{attribute 'pack_mode' := '1'} 
// ------------------------------------------------------------------------- 
//  SRCI Robot Library                                                
// ------------------------------------------------------------------------- 
//                                                                           
//  Object:      FreeDriveParCmd                                       
//  Author:      Thorsten Brach                                                
//  Date:        2024-06-22
//
//  Description:                                              
//   
//                                                                           
//  Copyright: 
//    (C) 2024 Thorsten Brach. All rights reserved                                                                                                                                            
//             Licensed under the MIT License.
//                                                                           
//  Disclaimer:                                                                           
//    This project is provided without any guarantee and can be used for   
//    private and commercial purposes. Any use is at the user’s 
//    own risk and responsibility.
//
// -------------------------------------------------------------------------
TYPE FreeDriveParCmd :
STRUCT
END_STRUCT
END_TYPE

{attribute 'pack_mode' := '1'} 
// ------------------------------------------------------------------------- 
//  SRCI Robot Library                                                
// ------------------------------------------------------------------------- 
//                                                                           
//  Object:      FreeDriveRecvData                                       
//  Author:      Thorsten Brach                                                
//  Date:        2024-06-22
//
//  Description:                                              
//   
//                                                                           
//  Copyright: 
//    (C) 2024 Thorsten Brach. All rights reserved                                                                                                                                            
//             Licensed under the MIT License.
//                                                                           
//  Disclaimer:                                                                           
//    This project is provided without any guarantee and can be used for   
//    private and commercial purposes. Any use is at the user’s 
//    own risk and responsibility.
//
// -------------------------------------------------------------------------
TYPE FreeDriveRecvData EXTENDS RspHeader :
STRUCT
  /// TRUE when function is exchanging data
  Enabled : BOOL;
END_STRUCT
END_TYPE

{attribute 'pack_mode' := '1'}
// ------------------------------------------------------------------------- 
//  SRCI Robot Library                                                
// ------------------------------------------------------------------------- 
//                                                                           
//  Object:      FreeDriveSendData                                       
//  Author:      Thorsten Brach                                                
//  Date:        2024-06-22
//
//  Description:                                              
//   
//                                                                           
//  Copyright: 
//    (C) 2024 Thorsten Brach. All rights reserved                                                                                                                                            
//             Licensed under the MIT License.
//                                                                           
//  Disclaimer:                                                                           
//    This project is provided without any guarantee and can be used for   
//    private and commercial purposes. Any use is at the user’s 
//    own risk and responsibility.
//
// -------------------------------------------------------------------------
TYPE FreeDriveSendData EXTENDS CmdHeader: 
STRUCT
  /// Set TRUE to activate "FreeDrive".
  Enable : BOOL;
END_STRUCT
END_TYPE

{attribute 'pack_mode' := '1'} 
// ------------------------------------------------------------------------- 
//  SRCI Robot Library                                                
// ------------------------------------------------------------------------- 
//                                                                           
//  Object:      MeasuringInputOutCmd                                       
//  Author:      Thorsten Brach                                                
//  Date:        2024-06-21
//
//  Description:                                              
//   
//                                                                           
//  Copyright: 
//    (C) 2024 Thorsten Brach. All rights reserved                                                                                                                                            
//             Licensed under the MIT License.
//                                                                           
//  Disclaimer:                                                                           
//    This project is provided without any guarantee and can be used for   
//    private and commercial purposes. Any use is at the user’s 
//    own risk and responsibility.
//
// -------------------------------------------------------------------------
TYPE MeasuringInputOutCmd :
STRUCT
  /// FB is returning a unique ID for the called measurement.
  MeasuringID        : UINT;
  /// Measured robot position value at the rising edge of the digital input in selected coordinate systems (see input parameters ToolNo and FrameNo).
  Measurings         : ARRAY[1..2] OF MeasuringInputResult;  
END_STRUCT
END_TYPE

{attribute 'pack_mode' := '1'} 
// ------------------------------------------------------------------------- 
//  SRCI Robot Library                                                
// ------------------------------------------------------------------------- 
//                                                                           
//  Object:      MeasuringInputParCmd                                       
//  Author:      Thorsten Brach                                                
//  Date:        2024-06-21
//
//  Description:                                              
//   
//                                                                           
//  Copyright: 
//    (C) 2024 Thorsten Brach. All rights reserved                                                                                                                                            
//             Licensed under the MIT License.
//                                                                           
//  Disclaimer:                                                                           
//    This project is provided without any guarantee and can be used for   
//    private and commercial purposes. Any use is at the user’s 
//    own risk and responsibility.
//
// -------------------------------------------------------------------------
TYPE MeasuringInputParCmd :
STRUCT
  /// Type of measurement (at least one option must be supported):
  MeasuringMode      : MeasuringIoMode;
  /// Specifies the desired digital input register. 
  /// More information about the different periphery register can be found in chapter 6.4
  Index              : USINT;
  ///Specifies the desired bit in the digital input register, that should be read. 
  /// More information about the different periphery register can be found in chapter 6.4.
  BitNumber          : USINT;
END_STRUCT
END_TYPE

{attribute 'pack_mode' := '1'} 
// ------------------------------------------------------------------------- 
//  SRCI Robot Library                                                
// ------------------------------------------------------------------------- 
//                                                                           
//  Object:      MeasuringInputRecvData                                       
//  Author:      Thorsten Brach                                                
//  Date:        2024-06-21
//
//  Description:                                              
//   
//                                                                           
//  Copyright: 
//    (C) 2024 Thorsten Brach. All rights reserved                                                                                                                                            
//             Licensed under the MIT License.
//                                                                           
//  Disclaimer:                                                                           
//    This project is provided without any guarantee and can be used for   
//    private and commercial purposes. Any use is at the user’s 
//    own risk and responsibility.
//
// -------------------------------------------------------------------------
TYPE MeasuringInputRecvData EXTENDS RspHeader :
STRUCT
  /// FB is returning a unique ID for the called measurement.
  MeasuringID        : UINT;
  /// Measured robot position value at the rising edge of the digital input in selected coordinate systems (see input parameters ToolNo and FrameNo).
  Measurings         : ARRAY[1..2] OF MeasuringInputResult;  
END_STRUCT
END_TYPE

{attribute 'pack_mode' := '1'}
// ------------------------------------------------------------------------- 
//  SRCI Robot Library                                                
// ------------------------------------------------------------------------- 
//                                                                           
//  Object:      MeasuringInputSendData                                       
//  Author:      Thorsten Brach                                                
//  Date:        2024-06-21
//
//  Description:                                              
//   
//                                                                           
//  Copyright: 
//    (C) 2024 Thorsten Brach. All rights reserved                                                                                                                                            
//             Licensed under the MIT License.
//                                                                           
//  Disclaimer:                                                                           
//    This project is provided without any guarantee and can be used for   
//    private and commercial purposes. Any use is at the user’s 
//    own risk and responsibility.
//
// -------------------------------------------------------------------------
TYPE MeasuringInputSendData EXTENDS CmdHeader:   
STRUCT
  /// Type of measurement (at least one option must be supported):
  MeasuringMode      : MeasuringIoMode;
  /// Specifies the desired digital input register. 
  /// More information about the different periphery register can be found in chapter 6.4
  Index              : USINT;
  ///Specifies the desired bit in the digital input register, that should be read. 
  /// More information about the different periphery register can be found in chapter 6.4.
  BitNumber          : USINT;
END_STRUCT
END_TYPE

{attribute 'pack_mode' := '1'} 
// ------------------------------------------------------------------------- 
//  SRCI Robot Library                                                
// ------------------------------------------------------------------------- 
//                                                                           
//  Object:      BrakeTestOutCmd                                       
//  Author:      Thorsten Brach                                                
//  Date:        2024-06-01
//
//  Description:                                              
//   
//                                                                           
//  Copyright: 
//    (C) 2024 Thorsten Brach. All rights reserved                                                                                                                                            
//             Licensed under the MIT License.
//                                                                           
//  Disclaimer:                                                                           
//    This project is provided without any guarantee and can be used for   
//    private and commercial purposes. Any use is at the user’s 
//    own risk and responsibility.
//
// -------------------------------------------------------------------------
TYPE OpenBrakeOutCmd :
STRUCT
  /// TRUE when "OpenBrake" is active.
  Enabled                   : BOOL;  
  /// Indicates the brake release status of the main robot axes.
  /// • TRUE: The brake of the axis is opened.
  /// • FALSE: The brake of the axis is closed.
  /// See Table 6-735 for bit assignment
  RobotAxesBrakeReleased    : RobotAxesFlags;
  /// Indicates the brake release status of the external robot axes.
  /// • TRUE: The brake of the axis is opened.
  /// • FALSE: The brake of the axis is closed/not supported
  /// See Table 6-735 for bit assignment
  ExternalAxesBrakeReleased : ExternalAxesFlags;
END_STRUCT
END_TYPE

{attribute 'pack_mode' := '1'} 
// ------------------------------------------------------------------------- 
//  SRCI Robot Library                                                
// ------------------------------------------------------------------------- 
//                                                                           
//  Object:      OpenBrakeParCmd                                       
//  Author:      Thorsten Brach                                                
//  Date:        2024-06-01
//
//  Description:                                              
//   
//                                                                           
//  Copyright: 
//    (C) 2024 Thorsten Brach. All rights reserved                                                                                                                                            
//             Licensed under the MIT License.
//                                                                           
//  Disclaimer:                                                                           
//    This project is provided without any guarantee and can be used for   
//    private and commercial purposes. Any use is at the user’s 
//    own risk and responsibility.
//
// -------------------------------------------------------------------------
TYPE OpenBrakeParCmd :
STRUCT
  /// Defines which brake of the robot axes must be released.
  /// • TRUE: Open the brake of the axis.
  /// • FALSE (default): Close the brake of the axis.
  RobotAxesBrakeRelease    : RobotAxesFlags;
  /// Defines which brake of the external robot axis must be released.
  /// • TRUE: Open the brake of the axis.
  /// • FALSE (default): Close the brake of the axis.
  /// See Table 6-676 for bit assignment.
  ExternalAxesBrakeRelease : ExternalAxesFlags;
END_STRUCT
END_TYPE

{attribute 'pack_mode' := '1'} 
// ------------------------------------------------------------------------- 
//  SRCI Robot Library                                                
// ------------------------------------------------------------------------- 
//                                                                           
//  Object:      BrakeTestRecvData                                       
//  Author:      Thorsten Brach                                                
//  Date:        2024-06-01
//
//  Description:                                              
//   
//                                                                           
//  Copyright: 
//    (C) 2024 Thorsten Brach. All rights reserved                                                                                                                                            
//             Licensed under the MIT License.
//                                                                           
//  Disclaimer:                                                                           
//    This project is provided without any guarantee and can be used for   
//    private and commercial purposes. Any use is at the user’s 
//    own risk and responsibility.
//
// -------------------------------------------------------------------------
TYPE OpenBrakeRecvData EXTENDS RspHeader :
STRUCT
  /// TRUE when "OpenBrake" is active.
  Enabled                   : BYTE;  
  /// Indicates the brake release status of the main robot axes.
  /// • TRUE: The brake of the axis is opened.
  /// • FALSE: The brake of the axis is closed.
  /// See Table 6-735 for bit assignment
  RobotAxesBrakeReleased    : BYTE;
  /// Indicates the brake release status of the external robot axes.
  /// • TRUE: The brake of the axis is opened.
  /// • FALSE: The brake of the axis is closed/not supported
  /// See Table 6-735 for bit assignment
  ExternalAxesBrakeReleased : BYTE;
END_STRUCT
END_TYPE

{attribute 'pack_mode' := '1'}
// ------------------------------------------------------------------------- 
//  SRCI Robot Library                                                
// ------------------------------------------------------------------------- 
//                                                                           
//  Object:      BrakeTestSendData                                       
//  Author:      Thorsten Brach                                                
//  Date:        2024-06-01
//
//  Description:                                              
//   
//                                                                           
//  Copyright: 
//    (C) 2024 Thorsten Brach. All rights reserved                                                                                                                                            
//             Licensed under the MIT License.
//                                                                           
//  Disclaimer:                                                                           
//    This project is provided without any guarantee and can be used for   
//    private and commercial purposes. Any use is at the user’s 
//    own risk and responsibility.
//
// -------------------------------------------------------------------------
TYPE OpenBrakeSendData EXTENDS CmdHeader:   
STRUCT
  /// Defines which brake of the robot axes must be released.
  /// • TRUE: Open the brake of the axis.
  /// • FALSE (default): Close the brake of the axis.
  RobotAxesBrakeRelease    : BYTE;
  /// Defines which brake of the external robot axis must be released.
  /// • TRUE: Open the brake of the axis.
  /// • FALSE (default): Close the brake of the axis.
  /// See Table 6-676 for bit assignment.
  ExternalAxesBrakeRelease : BYTE;
END_STRUCT
END_TYPE

{attribute 'pack_mode' := '1'} 
// ------------------------------------------------------------------------- 
//  SRCI Robot Library                                                
// ------------------------------------------------------------------------- 
//                                                                           
//  Object:      PathAccuracyModeOutCmd                                       
//  Author:      Thorsten Brach                                                
//  Date:        2024-06-22
//
//  Description:                                              
//   
//                                                                           
//  Copyright: 
//    (C) 2024 Thorsten Brach. All rights reserved                                                                                                                                            
//             Licensed under the MIT License.
//                                                                           
//  Disclaimer:                                                                           
//    This project is provided without any guarantee and can be used for   
//    private and commercial purposes. Any use is at the user’s 
//    own risk and responsibility.
//
// -------------------------------------------------------------------------
TYPE PathAccuracyModeOutCmd :
STRUCT
END_STRUCT
END_TYPE

{attribute 'pack_mode' := '1'} 
// ------------------------------------------------------------------------- 
//  SRCI Robot Library                                                
// ------------------------------------------------------------------------- 
//                                                                           
//  Object:      PathAccuracyModeParCmd                                       
//  Author:      Thorsten Brach                                                
//  Date:        2024-06-22
//
//  Description:                                              
//   
//                                                                           
//  Copyright: 
//    (C) 2024 Thorsten Brach. All rights reserved                                                                                                                                            
//             Licensed under the MIT License.
//                                                                           
//  Disclaimer:                                                                           
//    This project is provided without any guarantee and can be used for   
//    private and commercial purposes. Any use is at the user’s 
//    own risk and responsibility.
//
// -------------------------------------------------------------------------
TYPE PathAccuracyModeParCmd :
STRUCT
END_STRUCT
END_TYPE

{attribute 'pack_mode' := '1'} 
// ------------------------------------------------------------------------- 
//  SRCI Robot Library                                                
// ------------------------------------------------------------------------- 
//                                                                           
//  Object:      PathAccuracyModeRecvData                                       
//  Author:      Thorsten Brach                                                
//  Date:        2024-06-22
//
//  Description:                                              
//   
//                                                                           
//  Copyright: 
//    (C) 2024 Thorsten Brach. All rights reserved                                                                                                                                            
//             Licensed under the MIT License.
//                                                                           
//  Disclaimer:                                                                           
//    This project is provided without any guarantee and can be used for   
//    private and commercial purposes. Any use is at the user’s 
//    own risk and responsibility.
//
// -------------------------------------------------------------------------
TYPE PathAccuracyModeRecvData EXTENDS RspHeader :
STRUCT
  /// TRUE while PathAccuracyMode is active
  Enabled : BOOL;
END_STRUCT
END_TYPE

{attribute 'pack_mode' := '1'}
// ------------------------------------------------------------------------- 
//  SRCI Robot Library                                                
// ------------------------------------------------------------------------- 
//                                                                           
//  Object:      PathAccuracyModeSendData                                       
//  Author:      Thorsten Brach                                                
//  Date:        2024-06-22
//
//  Description:                                              
//   
//                                                                           
//  Copyright: 
//    (C) 2024 Thorsten Brach. All rights reserved                                                                                                                                            
//             Licensed under the MIT License.
//                                                                           
//  Disclaimer:                                                                           
//    This project is provided without any guarantee and can be used for   
//    private and commercial purposes. Any use is at the user’s 
//    own risk and responsibility.
//
// -------------------------------------------------------------------------
TYPE PathAccuracyModeSendData EXTENDS CmdHeader: 
STRUCT
  /// Set TRUE to activate monitoring of work areas
  Enable             : BOOL;
END_STRUCT
END_TYPE

{attribute 'pack_mode' := '1'} 
// ------------------------------------------------------------------------- 
//  SRCI Robot Library                                                
// ------------------------------------------------------------------------- 
//                                                                           
//  Object:      UnitMeasurementOutCmd                                       
//  Author:      Thorsten Brach                                                
//  Date:        2024-08-11
//
//  Description:                                              
//   
//                                                                           
//  Copyright: 
//    (C) 2024 Thorsten Brach. All rights reserved                                                                                                                                            
//             Licensed under the MIT License.
//                                                                           
//  Disclaimer:                                                                           
//    This project is provided without any guarantee and can be used for   
//    private and commercial purposes. Any use is at the user’s 
//    own risk and responsibility.
//
// -------------------------------------------------------------------------
TYPE ReadCallSubprogramCyclicOutCmd :
STRUCT
  /// Cyclic input data of subprogram
  Data : ARRAY[0..25] OF BYTE;
END_STRUCT
END_TYPE

{attribute 'pack_mode' := '1'} 
// ------------------------------------------------------------------------- 
//  SRCI Robot Library                                                
// ------------------------------------------------------------------------- 
//                                                                           
//  Object:      UnitMeasurementParCmd                                       
//  Author:      Thorsten Brach                                                
//  Date:        2024-08-11
//
//  Description:                                              
//   
//                                                                           
//  Copyright: 
//    (C) 2024 Thorsten Brach. All rights reserved                                                                                                                                            
//             Licensed under the MIT License.
//                                                                           
//  Disclaimer:                                                                           
//    This project is provided without any guarantee and can be used for   
//    private and commercial purposes. Any use is at the user’s 
//    own risk and responsibility.
//
// -------------------------------------------------------------------------
TYPE ReadCallSubprogramCyclicParCmd :
STRUCT
END_STRUCT
END_TYPE

{attribute 'pack_mode' := '1'} 
// ------------------------------------------------------------------------- 
//  SRCI Robot Library                                                
// ------------------------------------------------------------------------- 
//                                                                           
//  Object:      ShiftPositionOutCmd                                       
//  Author:      Thorsten Brach                                                
//  Date:        2024-06-22
//
//  Description:                                              
//   
//                                                                           
//  Copyright: 
//    (C) 2024 Thorsten Brach. All rights reserved                                                                                                                                            
//             Licensed under the MIT License.
//                                                                           
//  Disclaimer:                                                                           
//    This project is provided without any guarantee and can be used for   
//    private and commercial purposes. Any use is at the user’s 
//    own risk and responsibility.
//
// -------------------------------------------------------------------------
TYPE ShiftPositionOutCmd :
STRUCT
  /// Tool index
  TransformedPosition       : RobotCartesianPosition;  
END_STRUCT
END_TYPE

{attribute 'pack_mode' := '1'} 
// ------------------------------------------------------------------------- 
//  SRCI Robot Library                                                
// ------------------------------------------------------------------------- 
//                                                                           
//  Object:      ShiftPositionParCmd                                       
//  Author:      Thorsten Brach                                                
//  Date:        2024-06-22
//
//  Description:                                              
//   
//                                                                           
//  Copyright: 
//    (C) 2024 Thorsten Brach. All rights reserved                                                                                                                                            
//             Licensed under the MIT License.
//                                                                           
//  Disclaimer:                                                                           
//    This project is provided without any guarantee and can be used for   
//    private and commercial purposes. Any use is at the user’s 
//    own risk and responsibility.
//
// -------------------------------------------------------------------------
TYPE ShiftPositionParCmd :
STRUCT
  /// Define which method should be used to transform the position:
  Mode                      : TransformMode;
  /// Absolute coordinates of the position that will be transformed in the selected coordinate systems (see input parameter CoordinateSystem).
  Position                  : RobotCartesianPosition;
  /// Defines the reference frame ID to which the "Position" that will be transformed is relative.
  /// • 0: WCS (default)
  /// • 1..254: User frames
  FrameNo                   : USINT;
  /// Defines the reference frame ID to which the "TransformedPosition" should be relative.
  /// • 0: WCS (default)
  /// • 1..254: User frames
  TargetFrameNo             : USINT;
  /// Defines the frame data relevant for the transformation of the "Position". Relates to all "Mode" settings. 
  /// The parameter includes the Frame ID to which the origin of the shifting and rotation is relative and the cartesian position of the origin
  TransformationParameter_1 : FrameData;
  /// Relates to all "Mode" settings. Defines the enabled axis or plane as reference straight line or reference plain for the transformation
  TransformationParameter_2 : ReferenceElement;
  /// Defines the angle of rotation around the defined straight line. 
  /// Related to "Mode" with the setting "Rotate around Straight Line".
  RotationAngle             : REAL;  
END_STRUCT
END_TYPE

{attribute 'pack_mode' := '1'} 
// ------------------------------------------------------------------------- 
//  SRCI Robot Library                                                
// ------------------------------------------------------------------------- 
//                                                                           
//  Object:      ShiftPositionRecvData                                       
//  Author:      Thorsten Brach                                                
//  Date:        2024-06-22
//
//  Description:                                              
//   
//                                                                           
//  Copyright: 
//    (C) 2024 Thorsten Brach. All rights reserved                                                                                                                                            
//             Licensed under the MIT License.
//                                                                           
//  Disclaimer:                                                                           
//    This project is provided without any guarantee and can be used for   
//    private and commercial purposes. Any use is at the user’s 
//    own risk and responsibility.
//
// -------------------------------------------------------------------------
TYPE ShiftPositionRecvData EXTENDS RspHeader :
STRUCT
  /// Tool index
  TransformedPosition : RobotCartesianPosition;  
END_STRUCT
END_TYPE

{attribute 'pack_mode' := '1'}
// ------------------------------------------------------------------------- 
//  SRCI Robot Library                                                
// ------------------------------------------------------------------------- 
//                                                                           
//  Object:      ShiftPositionSendData                                       
//  Author:      Thorsten Brach                                                
//  Date:        2024-06-22
//
//  Description:                                              
//   
//                                                                           
//  Copyright: 
//    (C) 2024 Thorsten Brach. All rights reserved                                                                                                                                            
//             Licensed under the MIT License.
//                                                                           
//  Disclaimer:                                                                           
//    This project is provided without any guarantee and can be used for   
//    private and commercial purposes. Any use is at the user’s 
//    own risk and responsibility.
//
// -------------------------------------------------------------------------
TYPE ShiftPositionSendData EXTENDS CmdHeader: 
STRUCT
  /// Defines the frame data relevant for the transformation of the "Position". Relates to all "Mode" settings. 
  /// The parameter includes the Frame ID to which the origin of the shifting and rotation is relative and the cartesian position of the origin
  TransformationParameter_1 : FrameData;
  /// Relates to all "Mode" settings. Defines the enabled axis or plane as reference straight line or reference plain for the transformation
  TransformationParameter_2 : ReferenceElement;
  /// Defines the angle of rotation around the defined straight line. 
  /// Related to "Mode" with the setting "Rotate around Straight Line".
  RotationAngle             : REAL;
  /// Define which method should be used to transform the position:
  Mode                      : TransformMode;
  /// Defines the reference frame ID to which the "Position" that will be transformed is relative.
  /// • 0: WCS (default)
  /// • 1..254: User frames
  FrameNo                   : USINT;
  /// Defines the reference frame ID to which the "TransformedPosition" should be relative.
  /// • 0: WCS (default)
  /// • 1..254: User frames
  TargetFrameNo             : USINT;
  /// Absolute coordinates of the position that will be transformed in the selected coordinate systems (see input parameter CoordinateSystem).
  Position                  : RobotCartesianPosition;
END_STRUCT
END_TYPE

{attribute 'pack_mode' := '1'} 
// ------------------------------------------------------------------------- 
//  SRCI Robot Library                                                
// ------------------------------------------------------------------------- 
//                                                                           
//  Object:      SoftSwitchTcpOutCmd                                       
//  Author:      Thorsten Brach                                                
//  Date:        2024-06-30
//
//  Description:                                              
//   
//                                                                           
//  Copyright: 
//    (C) 2024 Thorsten Brach. All rights reserved                                                                                                                                            
//             Licensed under the MIT License.
//                                                                           
//  Disclaimer:                                                                           
//    This project is provided without any guarantee and can be used for   
//    private and commercial purposes. Any use is at the user’s 
//    own risk and responsibility.
//
// -------------------------------------------------------------------------
TYPE SoftSwitchTcpOutCmd :
STRUCT
  /// If TRUE, the RA is in a compliant movement.
  SoftMovement : BOOL;
END_STRUCT
END_TYPE

{attribute 'pack_mode' := '1'} 
// ------------------------------------------------------------------------- 
//  SRCI Robot Library                                                
// ------------------------------------------------------------------------- 
//                                                                           
//  Object:      SoftSwitchTcpParCmd                                       
//  Author:      Thorsten Brach                                                
//  Date:        2024-06-30
//
//  Description:                                              
//   
//                                                                           
//  Copyright: 
//    (C) 2024 Thorsten Brach. All rights reserved                                                                                                                                            
//             Licensed under the MIT License.
//                                                                           
//  Disclaimer:                                                                           
//    This project is provided without any guarantee and can be used for   
//    private and commercial purposes. Any use is at the user’s 
//    own risk and responsibility.
//
// -------------------------------------------------------------------------
TYPE SoftSwitchTcpParCmd :
STRUCT
  /// Defines type of reference coordinate system at which the robot can be moved in a compliant manner.
  ReferenceType       : ReferenceType;
  /// Index of tool or frame according to ReferenceType.
  /// • 0 (default): Flange/WS
  /// • 1..254: Tool/User frames
  ReferenceNo         : USINT;
  /// Relates to "LimitMode" with the setting "No limit defined". Defines for which cartesian axes the compliant motion is allowed. 
  /// If TRUE, the direction is enabled. Default value is FALSE. See Table 6-744 for bit assignment.
  CompliantAxes       : BYTE;
  /// Defines which parameters will limit the space, where the robot complies (at least one option must be supported)
  LimitMode           : LimitMode;
  /// Defines the type of the resistance force applied at the RA against the external force
  ResistanceForceMode : ResistanceForceMode;
  /// Relates to "ResistanceForceMode" with the setting "ResistanceForceTCP".
  /// Defines the resistance force level applied at the RA against the external force.
  /// • 0..99: Resistance is lower than robot vendor default. The lower the value, the easier the robot can be pushed away.
  /// • 100 (default): The value is aligned with the robot vendor-specific default value.
  /// • 101..200: Resistance is higher than robot vendor default. At maximum value "200" highest possible resistance against external force
  ResistanceForceTCP  : REAL;
  /// Relates to "ResistanceForceMode" with the setting "ResistanceForceAxis".
  /// Defines the resistance force level of the RA at the respective cartesian axis.
  ///  0..99: Resistance is lower than robot vendor default. The lower the value, the easier the robot can be pushed away.
  /// • 100 (default): The value is aligned with the robot vendor-specific default value.
  /// • 101..200: Resistance is higher than robot vendor default. At maximum value "200" highest possible resistance against external force.
  /// Index:
  /// • [0]: X-Axis O
  /// • [1]: Y-axis O
  /// • [2]: Z-axis O
  /// • [3]: RX-Direction O
  /// • [4]: RY-direction O
  /// • [5]: RZ-direction
  ResistanceForceAxis : ARRAY[0..5] OF REAL;
  /// Relates to "LimitMode" with the setting "Limit defined". 
  /// Limit values in the selected cartesian coordinate system (see input parameters ReferenceType and ReferenceNo).
  /// "0" is (default) the origin of the vector, the TCP position, at the start position of the robot.
  /// See Table 6-742 for the parameter index assignment.
  VectorData          : ARRAY[0..5] OF REAL;
END_STRUCT
END_TYPE

{attribute 'pack_mode' := '1'} 
// ------------------------------------------------------------------------- 
//  SRCI Robot Library                                                
// ------------------------------------------------------------------------- 
//                                                                           
//  Object:      SoftSwitchTcpRecvData                                       
//  Author:      Thorsten Brach                                                
//  Date:        2024-06-30
//
//  Description:                                              
//   
//                                                                           
//  Copyright: 
//    (C) 2024 Thorsten Brach. All rights reserved                                                                                                                                            
//             Licensed under the MIT License.
//                                                                           
//  Disclaimer:                                                                           
//    This project is provided without any guarantee and can be used for   
//    private and commercial purposes. Any use is at the user’s 
//    own risk and responsibility.
//
// -------------------------------------------------------------------------
TYPE SoftSwitchTcpRecvData EXTENDS RspHeader :
STRUCT
  /// If TRUE, the RA is in a compliant movement.
  SoftMovement : BOOL;  
END_STRUCT
END_TYPE

{attribute 'pack_mode' := '1'}
// ------------------------------------------------------------------------- 
//  SRCI Robot Library                                                
// ------------------------------------------------------------------------- 
//                                                                           
//  Object:      SoftSwitchTcpSendData                                       
//  Author:      Thorsten Brach                                                
//  Date:        2024-06-30
//
//  Description:                                              
//   
//                                                                           
//  Copyright: 
//    (C) 2024 Thorsten Brach. All rights reserved                                                                                                                                            
//             Licensed under the MIT License.
//                                                                           
//  Disclaimer:                                                                           
//    This project is provided without any guarantee and can be used for   
//    private and commercial purposes. Any use is at the user’s 
//    own risk and responsibility.
//
// -------------------------------------------------------------------------
TYPE SoftSwitchTcpSendData EXTENDS CmdHeader: 
STRUCT
  /// Defines which parameters will limit the space, where the robot complies (at least one option must be supported)
  LimitMode           : LimitMode;
  /// Relates to "LimitMode" with the setting "No limit defined". Defines for which cartesian axes the compliant motion is allowed. 
  /// If TRUE, the direction is enabled. Default value is FALSE. See Table 6-744 for bit assignment.
  CompliantAxes       : BYTE;
  /// Defines type of reference coordinate system at which the robot can be moved in a compliant manner.
  ReferenceType       : ReferenceType;  
  /// Index of tool or frame according to ReferenceType.
  /// • 0 (default): Flange/WS
  /// • 1..254: Tool/User frames
  ReferenceNo         : USINT;
  /// Relates to "ResistanceForceMode" with the setting "ResistanceForceTCP".
  /// Defines the resistance force level applied at the RA against the external force.
  /// • 0..99: Resistance is lower than robot vendor default. The lower the value, the easier the robot can be pushed away.
  /// • 100 (default): The value is aligned with the robot vendor-specific default value.
  /// • 101..200: Resistance is higher than robot vendor default. At maximum value "200" highest possible resistance against external force
  ResistanceForceTCP  : INT;
  /// Relates to "ResistanceForceMode" with the setting "ResistanceForceAxis".
  /// Defines the resistance force level of the RA at the respective cartesian axis.
  ///  0..99: Resistance is lower than robot vendor default. The lower the value, the easier the robot can be pushed away.
  /// • 100 (default): The value is aligned with the robot vendor-specific default value.
  /// • 101..200: Resistance is higher than robot vendor default. At maximum value "200" highest possible resistance against external force.
  /// Index:
  /// • [0]: X-Axis O
  /// • [1]: Y-axis O
  /// • [2]: Z-axis O
  /// • [3]: RX-Direction O
  /// • [4]: RY-direction O
  /// • [5]: RZ-direction
  ResistanceForceAxis : ARRAY[0..5] OF UINT;
  /// Relates to "LimitMode" with the setting "Limit defined". 
  /// Limit values in the selected cartesian coordinate system (see input parameters ReferenceType and ReferenceNo).
  /// "0" is (default) the origin of the vector, the TCP position, at the start position of the robot.
  /// See Table 6-742 for the parameter index assignment.
  VectorData          : ARRAY[0..5] OF REAL;
  /// Defines the type of the resistance force applied at the RA against the external force
  ResistanceForceMode : ResistanceForceMode;
END_STRUCT
END_TYPE

{attribute 'pack_mode' := '1'} 
// ------------------------------------------------------------------------- 
//  SRCI Robot Library                                                
// ------------------------------------------------------------------------- 
//                                                                           
//  Object:      StopSubprogramOutCmd                                       
//  Author:      Thorsten Brach                                                
//  Date:        2024-08-01
//
//  Description:                                              
//   
//                                                                           
//  Copyright: 
//    (C) 2024 Thorsten Brach. All rights reserved                                                                                                                                            
//             Licensed under the MIT License.
//                                                                           
//  Disclaimer:                                                                           
//    This project is provided without any guarantee and can be used for   
//    private and commercial purposes. Any use is at the user’s 
//    own risk and responsibility.
//
// -------------------------------------------------------------------------
TYPE StopSubprogramOutCmd :
STRUCT
  OriginID           : INT;
  /// Relates to ListenerID >0
  /// Number of successful trigger -based command invocations
  /// For more information refer to chapter 5.5.12.4.
  InvocationCounter  : USINT;
END_STRUCT
END_TYPE

{attribute 'pack_mode' := '1'} 
// ------------------------------------------------------------------------- 
//  SRCI Robot Library                                                
// ------------------------------------------------------------------------- 
//                                                                           
//  Object:      StopSubprogramParCmd                                       
//  Author:      Thorsten Brach                                                
//  Date:        2024-08-01
//
//  Description:                                              
//   
//                                                                           
//  Copyright: 
//    (C) 2024 Thorsten Brach. All rights reserved                                                                                                                                            
//             Licensed under the MIT License.
//                                                                           
//  Disclaimer:                                                                           
//    This project is provided without any guarantee and can be used for   
//    private and commercial purposes. Any use is at the user’s 
//    own risk and responsibility.
//
// -------------------------------------------------------------------------
TYPE StopSubprogramParCmd :
STRUCT
  /// Defines how target subprogram is defined
  StopMode          : StopMode;
  /// JobID or InstanceID of target subprogram according to selected StopMode
  /// • Refers to StopMode 0 (Stop via JobID) and 1 (Stop via InstanceID).
  /// • -1: Invalid (default)
  TargetID          : DINT;
  /// Defines the target sequence in which the command will be executed
  SequenceFlag      : SequenceFlag;
  /// ID of associated trigger function:
  /// • 0: No Trigger (default) - No trigger related behavior
  /// • >0: Triggero - Start executing when the trigger function with the identical EmitterID is triggered.
  /// Always positive.
  /// For more information, see chapter 5.5.12 Triggers
  ListenerID        : SINT;
  /// ID of Action that will be executed when this command is active
  /// • >0: Start Action - Start executing the Action function with the identical ListenerID.
  /// • <0: Stop Action  -  Stop executing the Action function with the identical ListenerID.
  /// • 0: No trigger (default)-  If no EmitterID is defined, the function will not trigger any Action during its execution
  /// For more information see section Triggers of this chapter or chapter 5.5.12.4.
  EmitterID          : ARRAY [0..3] OF SINT;  
END_STRUCT
END_TYPE

{attribute 'pack_mode' := '1'} 
// ------------------------------------------------------------------------- 
//  SRCI Robot Library                                                
// ------------------------------------------------------------------------- 
//                                                                           
//  Object:      StopSubprogramRecvData                                       
//  Author:      Thorsten Brach                                                
//  Date:        2024-08-01
//
//  Description:                                              
//   
//                                                                           
//  Copyright: 
//    (C) 2024 Thorsten Brach. All rights reserved                                                                                                                                            
//             Licensed under the MIT License.
//                                                                           
//  Disclaimer:                                                                           
//    This project is provided without any guarantee and can be used for   
//    private and commercial purposes. Any use is at the user’s 
//    own risk and responsibility.
//
// -------------------------------------------------------------------------
TYPE StopSubprogramRecvData EXTENDS RspHeader :
STRUCT
  /// Relates to ListenerID >0
  /// Number of successful trigger-based command invocations - For more information refer TO chapter 5.5.12.4
  InvocationCounter : USINT;  
  /// Reserve
  Reserve           : SINT;
  /// Unique system-generated ID of the "Action" when the function is triggered.
  /// • >0: The "Action" is started by the trigger funcrion with identical FollowID.
  /// • <0: The "Action" is stopped by the trigger function with identical FollowID.
  /// For more information see chapter 5.5.12.4 EmitterID, ListenerID, FollowID and OriginID
  OriginID          : INT;
END_STRUCT
END_TYPE

{attribute 'pack_mode' := '1'}
// ------------------------------------------------------------------------- 
//  SRCI Robot Library                                                
// ------------------------------------------------------------------------- 
//                                                                           
//  Object:      StopSubprogramSendData                                       
//  Author:      Thorsten Brach                                                
//  Date:        2024-08-01
//
//  Description:                                              
//   
//                                                                           
//  Copyright: 
//    (C) 2024 Thorsten Brach. All rights reserved                                                                                                                                            
//             Licensed under the MIT License.
//                                                                           
//  Disclaimer:                                                                           
//    This project is provided without any guarantee and can be used for   
//    private and commercial purposes. Any use is at the user’s 
//    own risk and responsibility.
//
// -------------------------------------------------------------------------
TYPE StopSubprogramSendData EXTENDS CmdHeader: 
STRUCT
  /// ID of Action that will be executed when this command is active
  /// • >0: Start Action - Start executing the Action function with the identical ListenerID.
  /// • <0: Stop Action  -  Stop executing the Action function with the identical ListenerID.
  /// • 0: No trigger (default)-  If no EmitterID is defined, the function will not trigger any Action during its execution
  /// For more information see section Triggers of this chapter or chapter 5.5.12.4.
  EmitterID          : ARRAY [0..3] OF SINT;  
  /// ID of associated trigger function:
  /// • 0: No Trigger (default) - No trigger related behavior
  /// • >0: Triggero - Start executing when the trigger function with the identical EmitterID is triggered.
  /// Always positive.
  /// For more information, see chapter 5.5.12 Triggers
  ListenerID        : SINT;
  /// Reserve
  Reserve           : BYTE;
  /// JobID or InstanceID of target subprogram according to selected StopMode
  /// • Refers to StopMode 0 (Stop via JobID) and 1 (Stop via InstanceID).
  /// • -1: Invalid (default)
  TargetID          : UINT;
  /// Defines how target subprogram is defined
  StopMode          : USINT;  
END_STRUCT
END_TYPE

{attribute 'pack_mode' := '1'} 
// ------------------------------------------------------------------------- 
//  SRCI Robot Library                                                
// ------------------------------------------------------------------------- 
//                                                                           
//  Object:      UnitMeasurementOutCmd                                       
//  Author:      Thorsten Brach                                                
//  Date:        2024-06-30
//
//  Description:                                              
//   
//                                                                           
//  Copyright: 
//    (C) 2024 Thorsten Brach. All rights reserved                                                                                                                                            
//             Licensed under the MIT License.
//                                                                           
//  Disclaimer:                                                                           
//    This project is provided without any guarantee and can be used for   
//    private and commercial purposes. Any use is at the user’s 
//    own risk and responsibility.
//
// -------------------------------------------------------------------------
TYPE UnitMeasurementOutCmd :
STRUCT
  /// TRUE, while the measurement is active.
  MeasurementActive : BOOL;
  /// Measurement result depending on the measurement type setting of the "MeasuringMode".
  Result            : REAL;
  /// Unique system-generated ID of the "Action" when the function is triggered.
  /// • >0: The "Action" is started by the trigger function with identical FollowID.
  /// • <0: The "Action" is stopped by the trigger function with identical FollowID.
  /// For more information see chapter 5.5.12.4 EmitterID, ListenerID, FollowID and OriginID
  OriginID           : INT;
  /// Relates to ListenerID >0
  /// Number of successful trigger -based command invocations
  /// For more information refer to chapter 5.5.12.4.
  InvocationCounter  : USINT;
END_STRUCT
END_TYPE

{attribute 'pack_mode' := '1'} 
// ------------------------------------------------------------------------- 
//  SRCI Robot Library                                                
// ------------------------------------------------------------------------- 
//                                                                           
//  Object:      UnitMeasurementParCmd                                       
//  Author:      Thorsten Brach                                                
//  Date:        2024-06-30
//
//  Description:                                              
//   
//                                                                           
//  Copyright: 
//    (C) 2024 Thorsten Brach. All rights reserved                                                                                                                                            
//             Licensed under the MIT License.
//                                                                           
//  Disclaimer:                                                                           
//    This project is provided without any guarantee and can be used for   
//    private and commercial purposes. Any use is at the user’s 
//    own risk and responsibility.
//
// -------------------------------------------------------------------------
TYPE UnitMeasurementParCmd :
STRUCT
  ///  Reaction type of measurement in relation to the trigger signal with the "ListenerID > 0" (at least one option must be supported):
  TriggerMode       : TriggerModeMeasurement;
  /// Relates to "TriggerMode" "No trigger related behavior".
  /// Set TRUE to start first measurement. Set TRUE again to receive new result data referring to previous rising edge of NewMeasurement.
  NewMeasurement    : BOOL;  
  /// Type of measurement (at least one option must be supported). 
 /// If the parameter is changed during the active measurement, the RC returns an error
  MeasuringMode     : MeasuringUnitMode;
  /// ID of the trigger function that may be triggered:
  /// • 0: Immediately (default). - Start executing THIS function immediately.
  /// • >0: Triggero Start executing when the trigger function with the identical EmitterID is called.
  /// For more information see chapter 5.5.12.4.
  ListenerID         : SINT;
END_STRUCT
END_TYPE

{attribute 'pack_mode' := '1'} 
// ------------------------------------------------------------------------- 
//  SRCI Robot Library                                                
// ------------------------------------------------------------------------- 
//                                                                           
//  Object:      UnitMeasurementRecvData                                       
//  Author:      Thorsten Brach                                                
//  Date:        2024-06-30
//
//  Description:                                              
//   
//                                                                           
//  Copyright: 
//    (C) 2024 Thorsten Brach. All rights reserved                                                                                                                                            
//             Licensed under the MIT License.
//                                                                           
//  Disclaimer:                                                                           
//    This project is provided without any guarantee and can be used for   
//    private and commercial purposes. Any use is at the user’s 
//    own risk and responsibility.
//
// -------------------------------------------------------------------------
TYPE UnitMeasurementRecvData EXTENDS RspHeader :
STRUCT
  /// Relates to ListenerID >0
  /// Number of successful trigger -based command invocations
  /// For more information refer to chapter 5.5.12.4.
  InvocationCounter : USINT;
  /// Reserve
  Reserve           : SINT;
  /// Unique system-generated ID of the "Action" when the function is triggered.
  /// • >0: The "Action" is started by the trigger function with identical FollowID.
  /// • <0: The "Action" is stopped by the trigger function with identical FollowID.
  /// For more information see chapter 5.5.12.4 EmitterID, ListenerID, FollowID and OriginID
  OriginID          : INT;
  /// Measurement result depending on the measurement type setting of the "MeasuringMode".
  Result            : REAL;
  /// TRUE, while the measurement is active.
  MeasurementActive : BOOL;
  /// TRUE, when new result data was received from the RC.
  ResultNo          : USINT;
END_STRUCT
END_TYPE

{attribute 'pack_mode' := '1'}
// ------------------------------------------------------------------------- 
//  SRCI Robot Library                                                
// ------------------------------------------------------------------------- 
//                                                                           
//  Object:      UnitMeasurementSendData                                       
//  Author:      Thorsten Brach                                                
//  Date:        2024-06-30
//
//  Description:                                              
//   
//                                                                           
//  Copyright: 
//    (C) 2024 Thorsten Brach. All rights reserved                                                                                                                                            
//             Licensed under the MIT License.
//                                                                           
//  Disclaimer:                                                                           
//    This project is provided without any guarantee and can be used for   
//    private and commercial purposes. Any use is at the user’s 
//    own risk and responsibility.
//
// -------------------------------------------------------------------------
TYPE UnitMeasurementSendData EXTENDS CmdHeader: 
STRUCT
  EmitterID     : ARRAY [0..3] OF SINT;
  /// ID of the trigger function that may be triggered:
  /// • 0: Immediately (default). - Start executing THIS function immediately.
  /// • >0: Triggero Start executing when the trigger function with the identical EmitterID is called.
  /// For more information see chapter 5.5.12.4.
  ListenerID    : SINT;
  /// Reserve
  Reserve       : BYTE;
  ///  Reaction type of measurement in relation to the trigger signal with the "ListenerID > 0" (at least one option must be supported):
  TriggerMode   : TriggerModeMeasurement;
  /// Relates to "TriggerMode" "No trigger related behavior".
  /// Set TRUE to start first measurement. Set TRUE again to receive new result data referring to previous rising edge of NewMeasurement.
  MeasurementNo : USINT;
  /// Type of measurement (at least one option must be supported). 
  /// If the parameter is changed during the active measurement, the RC returns an error
  MeasuringMode : MeasuringUnitMode;


END_STRUCT
END_TYPE

{attribute 'pack_mode' := '1'} 
// ------------------------------------------------------------------------- 
//  SRCI Robot Library                                                
// ------------------------------------------------------------------------- 
//                                                                           
//  Object:      UnitMeasurementOutCmd                                       
//  Author:      Thorsten Brach                                                
//  Date:        2024-08-11
//
//  Description:                                              
//   
//                                                                           
//  Copyright: 
//    (C) 2024 Thorsten Brach. All rights reserved                                                                                                                                            
//             Licensed under the MIT License.
//                                                                           
//  Disclaimer:                                                                           
//    This project is provided without any guarantee and can be used for   
//    private and commercial purposes. Any use is at the user’s 
//    own risk and responsibility.
//
// -------------------------------------------------------------------------
TYPE WriteCallSubprogramCyclicOutCmd :
STRUCT

END_STRUCT
END_TYPE

{attribute 'pack_mode' := '1'} 
// ------------------------------------------------------------------------- 
//  SRCI Robot Library                                                
// ------------------------------------------------------------------------- 
//                                                                           
//  Object:      UnitMeasurementParCmd                                       
//  Author:      Thorsten Brach                                                
//  Date:        2024-08-11
//
//  Description:                                              
//   
//                                                                           
//  Copyright: 
//    (C) 2024 Thorsten Brach. All rights reserved                                                                                                                                            
//             Licensed under the MIT License.
//                                                                           
//  Disclaimer:                                                                           
//    This project is provided without any guarantee and can be used for   
//    private and commercial purposes. Any use is at the user’s 
//    own risk and responsibility.
//
// -------------------------------------------------------------------------
TYPE WriteCallSubprogramCyclicParCmd :
STRUCT
  /// Cyclic input data of subprogram
  Data : ARRAY[0..25] OF BYTE;
END_STRUCT
END_TYPE

{attribute 'pack_mode' := '1'} 
// ------------------------------------------------------------------------- 
//  SRCI Robot Library                                                
// ------------------------------------------------------------------------- 
//                                                                           
//  Object:      MoveApproachDirectOutCmd                                       
//  Author:      Thorsten Brach                                                
//  Date:        2024-06-30
//
//  Description:                                              
//   
//                                                                           
//  Copyright: 
//    (C) 2024 Thorsten Brach. All rights reserved                                                                                                                                            
//             Licensed under the MIT License.
//                                                                           
//  Disclaimer:                                                                           
//    This project is provided without any guarantee and can be used for   
//    private and commercial purposes. Any use is at the user’s 
//    own risk and responsibility.
//
// -------------------------------------------------------------------------
TYPE MoveApproachDirectOutCmd :
STRUCT
  /// Distance-to-go of the current job.
  /// • -1: No valid value because move command is not yet active (valid values are pending) or not supported by RC
  /// • >0: Actual distance between current and target position
  /// •  0: Target position reached
  RemainingDistance  : REAL;
  /// Percentage of already traversed distance of current job.
  /// If not supported : • -1
  Progress           : REAL;
  /// Unique system-generated ID of the trigger function when the function is called by the user.
  /// For more information see chapter 5.5.12.4.
  FollowID           : DINT;  
END_STRUCT
END_TYPE

{attribute 'pack_mode' := '1'} 
// ------------------------------------------------------------------------- 
//  SRCI Robot Library                                                
// ------------------------------------------------------------------------- 
//                                                                           
//  Object:      MoveApproachDirectParCmd                                       
//  Author:      Thorsten Brach                                                
//  Date:        2024-06-30
//
//  Description:                                              
//   
//                                                                           
//  Copyright: 
//    (C) 2024 Thorsten Brach. All rights reserved                                                                                                                                            
//             Licensed under the MIT License.
//                                                                           
//  Disclaimer:                                                                           
//    This project is provided without any guarantee and can be used for   
//    private and commercial purposes. Any use is at the user’s 
//    own risk and responsibility.
//
// -------------------------------------------------------------------------
TYPE MoveApproachDirectParCmd :
STRUCT
  /// Absolute target coordinates in the selected coordinate system (see input parameters ToolNo and FrameNo).
  TargetPosition     : RobotCartesianPosition;
  /// Offset distance of auxiliary position from TargetPosition
  Offset             : AuxOffset;
  /// Defines type of reference coordinate system of the offset position
  ReferenceType      : ReferenceType;
  /// TCP velocity in % of nominal velocity
  /// •  <0%: (default) - Use default velocity
  /// •   0%:           - Use internal minimal velocity
  /// • 100%:           - Use maximal reference velocity
  /// See chapter 5.5.7 Robot dynamics
  VelocityRate       : REAL;
  /// Acceleration for movement in % of nominal acceleration
  /// •  <0%: (default) - Use default acceleration
  /// •   0%:           - Use internal minimal acceleration
  /// • 100%:           - Use maximal reference acceleration
  /// See chapter 5.5.7 Robot dynamics
  AccelerationRate   : REAL;
  /// Deceleration for movement in % of nominal deceleration
  /// •  <0%: (default) - Use default deceleration 
  /// •   0%:           - Use internal minimal deceleration
  /// • 100%:           - Use maximal reference deceleration
  /// See chapter 5.5.7 Robot dynamics
  DecelerationRate   : REAL;
  /// Jerk of the movement in % of nominal jerk
  /// •  <0%: (default) - Use default jerk
  /// •   0%:           - Use internal minimal jerk
  /// • 100%:           - Use maximal reference jerk
  /// See chapter 5.5.7 Robot dynamics
  JerkRate           : REAL;
  /// Index of tool
  /// •      0: Flange (default)
  /// • 1..254: Tool frames
  ToolNo             : USINT;
  /// Index of frame
  /// •      0: WCS (default)
  /// • 1..254: User frames
  FrameNo            : USINT;
  /// Parameter which determines the transition behavior at the end of the movement to be sent to the next command. 
  /// The user can choose a transition type between exact stop and different blend possibilities
  BlendingMode       : BlendingMode;
  /// Additional parameter for the blending mode, to define i.e. velocity limit (%) or blending radius
  BlendingParameter  : ARRAY [0..1] OF REAL := [10,0];
  /// Define blending sphere with radius around auxiliary position. For exact stop define AuxCornerDistance = 0
  AuxCornerDistance  : REAL;
  /// Parameter is used if it is greater than 0 (default)
  /// • Velocity input is ignored
  /// • Parameter defines the time for the movement to reach the target position
  /// Error is sent by the RC if the time cannot be kept
  MoveTime           : TIME;
  /// Parameter to describe how the orientation axes (RX, RY, RZ) will be interpolated during the movement
  OriMode            : OriMode;
  /// Defines the usage of the config byte inside the position according to Table 6-238
  ConfigMode         : ArmConfigParameter;
  /// Defines the usage of the TurnNumber byte inside the position.
  TurnMode           : TurnMode;
  /// Factor by which VelocityRate is multiplied to define the velocity for the second segment of the motion. Always positive.
  /// • 0: use the minimal velocity
  /// • 1: use the velocity set with VelocityRate 
  /// Input values below 1 to reduce velocity, 
  /// Input values above 1 to increase velocity.
  /// See chapter 5.5.7 Robot dynamics
  VelocityCoefficient: REAL;
  /// Set TRUE to allow manipulation of this move command through superimposing functions.
  /// For more information see chapter 5.5.9.5
  Manipulation       : BOOL;
  /// ID of Action that will be executed when this command is active
  /// • >0: Start Action - Start executing the Action function with the identical ListenerID.
  /// • <0: Stop Action  -  Stop executing the Action function with the identical ListenerID.
  /// • 0: No trigger (default)-  If no EmitterID is defined, the function will not trigger any Action during its execution
  /// For more information see section Triggers of this chapter or chapter 5.5.12.4.
  EmitterID          : ARRAY [0..3] OF SINT;
END_STRUCT
END_TYPE

{attribute 'pack_mode' := '1'} 
// ------------------------------------------------------------------------- 
//  SRCI Robot Library                                                
// ------------------------------------------------------------------------- 
//                                                                           
//  Object:      MoveApproachDirectRecvData                                       
//  Author:      Thorsten Brach                                                
//  Date:        2024-06-30
//
//  Description:                                              
//   
//                                                                           
//  Copyright: 
//    (C) 2024 Thorsten Brach. All rights reserved                                                                                                                                            
//             Licensed under the MIT License.
//                                                                           
//  Disclaimer:                                                                           
//    This project is provided without any guarantee and can be used for   
//    private and commercial purposes. Any use is at the user’s 
//    own risk and responsibility.
//
// -------------------------------------------------------------------------
TYPE MoveApproachDirectRecvData EXTENDS RspHeader :
STRUCT
  /// Relates to ListenerID >0
  /// Number of successful trigger-based command invocations - For more information refer TO chapter 5.5.12.4
  InvocationCounter : USINT;  
  /// Reserve
  Reserve           : SINT;
  /// Unique system-generated ID of the "Action" when the function is triggered.
  /// • >0: The "Action" is started by the trigger funcrion with identical FollowID.
  /// • <0: The "Action" is stopped by the trigger function with identical FollowID.
  /// For more information see chapter 5.5.12.4 EmitterID, ListenerID, FollowID and OriginID
  OriginID          : INT;
  /// Percentage of already traversed distance of current job.
  /// If not supported : • -1
  Progress          : UINT;
  /// Distance-to-go of the current job.
  /// • -1: No valid value because move command is not yet active (valid values are pending) or not supported by RC
  /// • >0: Actual distance between current and target position
  /// •  0: Target position reached
  RemainingDistance : REAL;
END_STRUCT
END_TYPE

{attribute 'pack_mode' := '1'}
// ------------------------------------------------------------------------- 
//  SRCI Robot Library                                                
// ------------------------------------------------------------------------- 
//                                                                           
//  Object:      MoveApproachDirectSendData                                       
//  Author:      Thorsten Brach                                                
//  Date:        2024-06-30
//
//  Description:                                              
//   
//                                                                           
//  Copyright: 
//    (C) 2024 Thorsten Brach. All rights reserved                                                                                                                                            
//             Licensed under the MIT License.
//                                                                           
//  Disclaimer:                                                                           
//    This project is provided without any guarantee and can be used for   
//    private and commercial purposes. Any use is at the user’s 
//    own risk and responsibility.
//
// -------------------------------------------------------------------------
TYPE MoveApproachDirectSendData EXTENDS CmdHeader: 
STRUCT
  /// ID of Action that will be executed when this command is active
  /// • >0: Start Action - Start executing the Action function with the identical ListenerID.
  /// • <0: Stop Action  -  Stop executing the Action function with the identical ListenerID.
  /// • 0: No trigger (default)-  If no EmitterID is defined, the function will not trigger any Action during its execution
  /// For more information see section Triggers of this chapter or chapter 5.5.12.4.
  EmitterID          : ARRAY [0..3] OF SINT;
  /// ID of the trigger function that may be triggered:
  /// • 0: Immediately (default). - Start executing THIS function immediately.
  /// • >0: Triggero Start executing when the trigger function with the identical EmitterID is called.
  /// For more information see chapter 5.5.12.4.
  ListenerID         : SINT;
  /// Reserve
  Reserve            : BYTE;
  /// TCP velocity in % of nominal velocity
  /// •  <0%: (default) - Use default velocity
  /// •   0%:           - Use internal minimal velocity
  /// • 100%:           - Use maximal reference velocity
  /// See chapter 5.5.7 Robot dynamics
  VelocityRate       : UINT;  
  /// Acceleration for movement in % of nominal acceleration
  /// •  <0%: (default) - Use default acceleration
  /// •   0%:           - Use internal minimal acceleration
  /// • 100%:           - Use maximal reference acceleration
  /// See chapter 5.5.7 Robot dynamics
  AccelerationRate   : UINT;
  /// Deceleration for movement in % of nominal deceleration
  /// •  <0%: (default) - Use default deceleration 
  /// •   0%:           - Use internal minimal deceleration
  /// • 100%:           - Use maximal reference deceleration
  /// See chapter 5.5.7 Robot dynamics
  DecelerationRate   : UINT;
  /// Jerk of the movement in % of nominal jerk
  /// •  <0%: (default) - Use default jerk
  /// •   0%:           - Use internal minimal jerk
  /// • 100%:           - Use maximal reference jerk
  /// See chapter 5.5.7 Robot dynamics
  JerkRate           : UINT;
  /// Index of tool
  /// •      0: Flange (default)
  /// • 1..254: Tool frames
  ToolNo             : USINT;
  /// Index of frame
  /// •      0: WCS (default)
  /// • 1..254: User frames
  FrameNo            : USINT;
  /// Parameter which determines the transition behavior at the end of the movement to be sent to the next command. 
  /// The user can choose a transition type between exact stop and different blend possibilities
  BlendingMode       : BlendingMode;
  /// Parameter to describe how the orientation axes (RX, RY, RZ) will be interpolated during the movement
  OriMode            : OriMode;
  /// Additional parameter for the blending mode, to define i.e. velocity limit (%) or blending radius
  BlendingParameter  : ARRAY [0..1] OF REAL := [10,0];
  /// Absolute target coordinates in the selected coordinate system (see input parameters ToolNo and FrameNo).
  TargetPosition     : RobotCartesianPosition;
  /// Offset distance of auxiliary position from TargetPosition
  Offset             : AuxOffset;
  /// Define blending sphere with radius around auxiliary position. For exact stop define AuxCornerDistance = 0
  AuxCornerDistance  : REAL;
  /// Factor by which VelocityRate is multiplied to define the velocity for the second segment of the motion. Always positive.
  /// • 0: use the minimal velocity
  /// • 1: use the velocity set with VelocityRate 
  /// Input values below 1 to reduce velocity, 
  /// Input values above 1 to increase velocity.
  /// See chapter 5.5.7 Robot dynamics
  VelocityCoefficient: REAL;
  /// Set TRUE to allow manipulation of this move command through superimposing functions.
  /// For more information see chapter 5.5.9.5
  Manipulation       : BOOL;
  /// Defines the usage of the config byte inside the position according to Table 6-238
  ConfigMode         :  ARRAY[0..1] OF BYTE;
  /// Defines the usage of the TurnNumber byte inside the position.
  TurnMode           : TurnMode;
  /// Defines type of reference coordinate system of the offset position
  ReferenceType      : ReferenceType;
  /// Parameter is used if it is greater than 0 (default)
  /// • Velocity input is ignored
  /// • Parameter defines the time for the movement to reach the target position
  /// Error is sent by the RC if the time cannot be kept
  MoveTime           : UINT;
END_STRUCT
END_TYPE

{attribute 'pack_mode' := '1'} 
// ------------------------------------------------------------------------- 
//  SRCI Robot Library                                                
// ------------------------------------------------------------------------- 
//                                                                           
//  Object:      MoveApproachLinearOutCmd                                       
//  Author:      Thorsten Brach                                                
//  Date:        2024-06-30
//
//  Description:                                              
//   
//                                                                           
//  Copyright: 
//    (C) 2024 Thorsten Brach. All rights reserved                                                                                                                                            
//             Licensed under the MIT License.
//                                                                           
//  Disclaimer:                                                                           
//    This project is provided without any guarantee and can be used for   
//    private and commercial purposes. Any use is at the user’s 
//    own risk and responsibility.
//
// -------------------------------------------------------------------------
TYPE MoveApproachLinearOutCmd :
STRUCT
  /// Distance-to-go of the current job.
  /// • -1: No valid value because move command is not yet active (valid values are pending) or not supported by RC
  /// • >0: Actual distance between current and target position
  /// •  0: Target position reached
  RemainingDistance  : REAL;
  /// Percentage of already traversed distance of current job.
  /// If not supported : • -1
  Progress           : REAL;
  /// Unique system-generated ID of the trigger function when the function is called by the user.
  /// For more information see chapter 5.5.12.4.
  FollowID           : DINT;  
END_STRUCT
END_TYPE

{attribute 'pack_mode' := '1'} 
// ------------------------------------------------------------------------- 
//  SRCI Robot Library                                                
// ------------------------------------------------------------------------- 
//                                                                           
//  Object:      MoveApproachLinearParCmd                                       
//  Author:      Thorsten Brach                                                
//  Date:        2024-06-30
//
//  Description:                                              
//   
//                                                                           
//  Copyright: 
//    (C) 2024 Thorsten Brach. All rights reserved                                                                                                                                            
//             Licensed under the MIT License.
//                                                                           
//  Disclaimer:                                                                           
//    This project is provided without any guarantee and can be used for   
//    private and commercial purposes. Any use is at the user’s 
//    own risk and responsibility.
//
// -------------------------------------------------------------------------
TYPE MoveApproachLinearParCmd :
STRUCT
  /// Absolute target coordinates in the selected coordinate system (see input parameters ToolNo and FrameNo).
  TargetPosition     : RobotCartesianPosition;
  /// Offset distance of auxiliary position from TargetPosition
  Offset             : AuxOffset;
  /// Defines type of reference coordinate system of the offset position
  ReferenceType      : ReferenceType;
  /// TCP velocity in % of nominal velocity
  /// •  <0%: (default) - Use default velocity
  /// •   0%:           - Use internal minimal velocity
  /// • 100%:           - Use maximal reference velocity
  /// See chapter 5.5.7 Robot dynamics
  VelocityRate       : REAL;
  /// Acceleration for movement in % of nominal acceleration
  /// •  <0%: (default) - Use default acceleration
  /// •   0%:           - Use internal minimal acceleration
  /// • 100%:           - Use maximal reference acceleration
  /// See chapter 5.5.7 Robot dynamics
  AccelerationRate   : REAL;
  /// Deceleration for movement in % of nominal deceleration
  /// •  <0%: (default) - Use default deceleration 
  /// •   0%:           - Use internal minimal deceleration
  /// • 100%:           - Use maximal reference deceleration
  /// See chapter 5.5.7 Robot dynamics
  DecelerationRate   : REAL;
  /// Jerk of the movement in % of nominal jerk
  /// •  <0%: (default) - Use default jerk
  /// •   0%:           - Use internal minimal jerk
  /// • 100%:           - Use maximal reference jerk
  /// See chapter 5.5.7 Robot dynamics
  JerkRate           : REAL;
  /// Index of tool
  /// •      0: Flange (default)
  /// • 1..254: Tool frames
  ToolNo             : USINT;
  /// Index of frame
  /// •      0: WCS (default)
  /// • 1..254: User frames
  FrameNo            : USINT;
  /// Parameter which determines the transition behavior at the end of the movement to be sent to the next command. 
  /// The user can choose a transition type between exact stop and different blend possibilities
  BlendingMode       : BlendingMode;
  /// Additional parameter for the blending mode, to define i.e. velocity limit (%) or blending radius
  BlendingParameter  : ARRAY [0..1] OF REAL := [10,0];
  /// Define blending sphere with radius around auxiliary position. For exact stop define AuxCornerDistance = 0
  AuxCornerDistance  : REAL;
  /// Parameter is used if it is greater than 0 (default)
  /// • Velocity input is ignored
  /// • Parameter defines the time for the movement to reach the target position
  /// Error is sent by the RC if the time cannot be kept
  MoveTime           : TIME;
  /// Parameter to describe how the orientation axes (RX, RY, RZ) will be interpolated during the movement
  OriMode            : OriMode;
  /// Defines the usage of the config byte inside the position according to Table 6-238
  ConfigMode         : ArmConfigParameter;
  /// Defines the usage of the TurnNumber byte inside the position.
  TurnMode           : TurnMode;
  /// Factor by which VelocityRate is multiplied to define the velocity for the second segment of the motion. Always positive.
  /// • 0: use the minimal velocity
  /// • 1: use the velocity set with VelocityRate 
  /// Input values below 1 to reduce velocity, 
  /// Input values above 1 to increase velocity.
  /// See chapter 5.5.7 Robot dynamics
  VelocityCoefficient: REAL;
  /// Set TRUE to allow manipulation of this move command through superimposing functions.
  /// For more information see chapter 5.5.9.5
  Manipulation       : BOOL;
  /// ID of Action that will be executed when this command is active
  /// • >0: Start Action - Start executing the Action function with the identical ListenerID.
  /// • <0: Stop Action  -  Stop executing the Action function with the identical ListenerID.
  /// • 0: No trigger (default)-  If no EmitterID is defined, the function will not trigger any Action during its execution
  /// For more information see section Triggers of this chapter or chapter 5.5.12.4.
  EmitterID          : ARRAY [0..3] OF SINT;
END_STRUCT
END_TYPE

{attribute 'pack_mode' := '1'} 
// ------------------------------------------------------------------------- 
//  SRCI Robot Library                                                
// ------------------------------------------------------------------------- 
//                                                                           
//  Object:      MoveApproachLinearRecvData                                       
//  Author:      Thorsten Brach                                                
//  Date:        2024-06-30
//
//  Description:                                              
//   
//                                                                           
//  Copyright: 
//    (C) 2024 Thorsten Brach. All rights reserved                                                                                                                                            
//             Licensed under the MIT License.
//                                                                           
//  Disclaimer:                                                                           
//    This project is provided without any guarantee and can be used for   
//    private and commercial purposes. Any use is at the user’s 
//    own risk and responsibility.
//
// -------------------------------------------------------------------------
TYPE MoveApproachLinearRecvData EXTENDS RspHeader :
STRUCT
  /// Relates to ListenerID >0
  /// Number of successful trigger-based command invocations - For more information refer TO chapter 5.5.12.4
  InvocationCounter : USINT;  
  /// Reserve
  Reserve           : SINT;
  /// Unique system-generated ID of the "Action" when the function is triggered.
  /// • >0: The "Action" is started by the trigger funcrion with identical FollowID.
  /// • <0: The "Action" is stopped by the trigger function with identical FollowID.
  /// For more information see chapter 5.5.12.4 EmitterID, ListenerID, FollowID and OriginID
  OriginID          : INT;
  /// Percentage of already traversed distance of current job.
  /// If not supported : • -1
  Progress          : UINT;
  /// Distance-to-go of the current job.
  /// • -1: No valid value because move command is not yet active (valid values are pending) or not supported by RC
  /// • >0: Actual distance between current and target position
  /// •  0: Target position reached
  RemainingDistance : REAL;  
END_STRUCT
END_TYPE

{attribute 'pack_mode' := '1'}
// ------------------------------------------------------------------------- 
//  SRCI Robot Library                                                
// ------------------------------------------------------------------------- 
//                                                                           
//  Object:      MoveApproachLinearSendData                                       
//  Author:      Thorsten Brach                                                
//  Date:        2024-06-30
//
//  Description:                                              
//   
//                                                                           
//  Copyright: 
//    (C) 2024 Thorsten Brach. All rights reserved                                                                                                                                            
//             Licensed under the MIT License.
//                                                                           
//  Disclaimer:                                                                           
//    This project is provided without any guarantee and can be used for   
//    private and commercial purposes. Any use is at the user’s 
//    own risk and responsibility.
//
// -------------------------------------------------------------------------
TYPE MoveApproachLinearSendData EXTENDS CmdHeader: 
STRUCT
/// ID of Action that will be executed when this command is active
  /// • >0: Start Action - Start executing the Action function with the identical ListenerID.
  /// • <0: Stop Action  -  Stop executing the Action function with the identical ListenerID.
  /// • 0: No trigger (default)-  If no EmitterID is defined, the function will not trigger any Action during its execution
  /// For more information see section Triggers of this chapter or chapter 5.5.12.4.
  EmitterID          : ARRAY [0..3] OF SINT;
  /// ID of the trigger function that may be triggered:
  /// • 0: Immediately (default). - Start executing THIS function immediately.
  /// • >0: Triggero Start executing when the trigger function with the identical EmitterID is called.
  /// For more information see chapter 5.5.12.4.
  ListenerID         : SINT;
  /// Reserve
  Reserve            : BYTE;
  /// TCP velocity in % of nominal velocity
  /// •  <0%: (default) - Use default velocity
  /// •   0%:           - Use internal minimal velocity
  /// • 100%:           - Use maximal reference velocity
  /// See chapter 5.5.7 Robot dynamics
  VelocityRate       : UINT;  
  /// Acceleration for movement in % of nominal acceleration
  /// •  <0%: (default) - Use default acceleration
  /// •   0%:           - Use internal minimal acceleration
  /// • 100%:           - Use maximal reference acceleration
  /// See chapter 5.5.7 Robot dynamics
  AccelerationRate   : UINT;
  /// Deceleration for movement in % of nominal deceleration
  /// •  <0%: (default) - Use default deceleration 
  /// •   0%:           - Use internal minimal deceleration
  /// • 100%:           - Use maximal reference deceleration
  /// See chapter 5.5.7 Robot dynamics
  DecelerationRate   : UINT;
  /// Jerk of the movement in % of nominal jerk
  /// •  <0%: (default) - Use default jerk
  /// •   0%:           - Use internal minimal jerk
  /// • 100%:           - Use maximal reference jerk
  /// See chapter 5.5.7 Robot dynamics
  JerkRate           : UINT;
  /// Index of tool
  /// •      0: Flange (default)
  /// • 1..254: Tool frames
  ToolNo             : USINT;
  /// Index of frame
  /// •      0: WCS (default)
  /// • 1..254: User frames
  FrameNo            : USINT;
  /// Parameter which determines the transition behavior at the end of the movement to be sent to the next command. 
  /// The user can choose a transition type between exact stop and different blend possibilities
  BlendingMode       : BlendingMode;
  /// Parameter to describe how the orientation axes (RX, RY, RZ) will be interpolated during the movement
  OriMode            : OriMode;
  /// Additional parameter for the blending mode, to define i.e. velocity limit (%) or blending radius
  BlendingParameter  : ARRAY [0..1] OF REAL := [10,0];
  /// Absolute target coordinates in the selected coordinate system (see input parameters ToolNo and FrameNo).
  TargetPosition     : RobotCartesianPosition;
  /// Offset distance of auxiliary position from TargetPosition
  Offset             : AuxOffset;
  /// Define blending sphere with radius around auxiliary position. For exact stop define AuxCornerDistance = 0
  AuxCornerDistance  : REAL;
  /// Factor by which VelocityRate is multiplied to define the velocity for the second segment of the motion. Always positive.
  /// • 0: use the minimal velocity
  /// • 1: use the velocity set with VelocityRate 
  /// Input values below 1 to reduce velocity, 
  /// Input values above 1 to increase velocity.
  /// See chapter 5.5.7 Robot dynamics
  VelocityCoefficient: REAL;
  /// Set TRUE to allow manipulation of this move command through superimposing functions.
  /// For more information see chapter 5.5.9.5
  Manipulation       : BOOL;
  /// Defines the usage of the config byte inside the position according to Table 6-238
  ConfigMode         :  ARRAY[0..1] OF BYTE;
  /// Defines the usage of the TurnNumber byte inside the position.
  TurnMode           : TurnMode;
  /// Defines type of reference coordinate system of the offset position
  ReferenceType      : ReferenceType;
  /// Parameter is used if it is greater than 0 (default)
  /// • Velocity input is ignored
  /// • Parameter defines the time for the movement to reach the target position
  /// Error is sent by the RC if the time cannot be kept
  MoveTime           : UINT;  
END_STRUCT
END_TYPE

